FUNCTION F_Trim : STRING
VAR_INPUT
    s : STRING;
END_VAR

END_FUNCTION

(* stored: Version 1.1.0.1
   POU F_Trim: Id {76050ca4-0bf3-47fd-b12d-3a4ea2bd6466}, SpecialFunc None *)
